// TwinCAT 3 PLC project tc_mot_example
// ProgramVersion: 3.1.4022.7
// CompilerDefines: L
// libraries:
//   LCLS General, * (SLAC)
//   lcls-twincat-motion, * (SLAC)
//   lcls2-cc-lib, * (SLAC)
//   PMPS, * (SLAC - LCLS)
//   Tc2_SerialCom, * (Beckhoff Automation GmbH)
//   Tc2_Standard, * (Beckhoff Automation GmbH)
//   Tc2_System, * (Beckhoff Automation GmbH)
//   Tc3_Module, * (Beckhoff Automation GmbH)
// project tree:
//   GVLs/ GVL.TcGVL
//   / PlcTask.TcTTO (not stored)
//   POUs/ Main.TcPOU
// real-time tasks:
//   TASK PlcTask: cycle T#10ms, priority 20, ADS port 350
// motion (NC):
// variable links:
//   tc_mot_example Instance <-> NC-Task 1 SAF/Axes/Example 1 Simulated Working
//     PlcTask Inputs/Main.M1.Axis.NcToPlc <-> Outputs/ToPlc
//     PlcTask Outputs/Main.M1.Axis.PlcToNc <-> Inputs/FromPlc
//   tc_mot_example Instance <-> NC-Task 1 SAF/Axes/Example 2 Simulated Broken
//     PlcTask Inputs/Main.M2.Axis.NcToPlc <-> Outputs/ToPlc
//     PlcTask Outputs/Main.M2.Axis.PlcToNc <-> Inputs/FromPlc
//   tc_mot_example Instance <-> NC-Task 1 SAF/Axes/Example 3 Simulated Limits
//     PlcTask Inputs/Main.M3.Axis.NcToPlc <-> Outputs/ToPlc
//     PlcTask Outputs/Main.M3.Axis.PlcToNc <-> Inputs/FromPlc

// ---- GVLs/GVL.TcGVL
{attribute 'qualified_only'}
VAR_GLOBAL
    fbArbiter: FB_Arbiter(1);
    fbFastFaultOutput1: FB_HardwareFFOutput := (bAutoReset := TRUE, i_sNetID := '172.21.148.148.1.1');
END_VAR

// ---- POUs/Main.TcPOU
PROGRAM Main
VAR
    // Simulated motor that is always allowed to move
    {attribute 'pytmc' := '
        pv: PLC:TST:MOT:SIM:01
        field: DESC Simulated Working Motor
    '}
    M1: DUT_MotionStage;
    fbMotion1: FB_MotionStageSim;

    // Simulated motor that is never allowed to move
    {attribute 'pytmc' := '
        pv: PLC:TST:MOT:SIM:02
        field: DESC Simulated Broken Motor
    '}
    M2: DUT_MotionStage;
    fbMotion2: FB_MotionStage;

    // Simulated motor with limits at 0 and 100
    {attribute 'pytmc' := '
        pv: PLC:TST:MOT:SIM:03
        field: DESC Simulated Working Motor With Limits
    '}
    M3: DUT_MotionStage;
    fbMotion3: FB_MotionStage;


    {attribute 'pytmc' := '
        pv: PLC:TST:MOT:SIM:XPIM
        io: io
    '}
    fbIM1L0: FB_XPIM;
    stEL6In AT %I*: EL6InData22b;
    stEL6Out AT %Q*: EL6OutData22b;
    bInit: BOOL := TRUE;

    fbArbiterIO: FB_SubSysToArbiter_IO;
END_VAR

// fbMotion1(stMotionStage := M1);
// fbMotion2(stMotionStage := M2);
// fbMotion3(stMotionStage := M3);
// M3.bHardwareEnable := TRUE;
// M3.bPowerSelf := TRUE;
M3.bLimitForwardEnable := M3.Axis.NcToPlc.ActPos < 99.7;
M3.bLimitBackwardEnable := M3.Axis.NcToPlc.ActPos > 0.2;

IF bInit THEN
    fbIM1L0.stOut.fPosition := 0;
    fbIM1L0.stOut.bUseRawCounts := FALSE;
    fbIM1L0.stOut.stPMPS.sPmpsState := 'IM1K0-XTES-OUT';
    fbIM1L0.stOut.bValid := TRUE;
    fbIM1L0.stYag.fPosition := -86.65;
    fbIM1L0.stYag.bUseRawCounts := FALSE;
    fbIM1L0.stYag.stPMPS.sPmpsState := 'IM1K0-XTES-YAG';
    fbIM1L0.stYag.bValid := TRUE;
    fbIM1L0.stDiamond.fPosition := -56.65;
    fbIM1L0.stDiamond.bUseRawCounts := FALSE;
    fbIM1L0.stDiamond.stPMPS.sPmpsState := 'IM1K0-XTES-DIAMOND';
    fbIM1L0.stDiamond.bValid := TRUE;
    fbIM1L0.stReticle.fPosition := -26.65;
    fbIM1L0.stReticle.bUseRawCounts := FALSE;
    fbIM1L0.stReticle.stPMPS.sPmpsState := 'IM1K0-XTES-RETICLE';
    fbIM1L0.stReticle.bValid := TRUE;
    bInit := FALSE;
END_IF

fbIM1L0(
    fbArbiter := GVL.fbArbiter,
    fbFFHWO := GVL.fbFastFaultOutput1,
    stYStage := M1,
    stZoomStage := M2,
    stFocusStage := M3,
    stEl6In := stEL6In,
    stEl6Out := stEl6Out,
    sPmpsDeviceName := 'IM1K0-XTES',
    sTransitionKey:='IM1K0-MOVING',
);

MOTION_GVL.fbStandardPMPSDB(
    io_fbFFHWO:=GVL.fbFastFaultOutput1,
    bEnable:=TRUE,
    sPLCName:='tst-motion',
);
GVL.fbFastFaultOutput1.Execute();
fbArbiterIO(
    Arbiter:=GVL.fbArbiter,
    fbFFHWO:=GVL.fbFastFaultOutput1);

END_PROGRAM
